{attribute 'strict'}
TYPE E_StewartMode :
(
	eIDLE := 0,
	eTRANSITION,
	eSIMULATION,
	eXBOX,
	eERROR
);
END_TYPE

(* stored: Version 1.1.0.1, ProductVersion 3.1.4022.7
   DUT E_StewartMode: Id {bb43455b-ecbe-48a4-ba16-432357bafc03} *)
